// TIA Portal project "Oefening 9" (V14)

(* hardware
DEVICE "S7300/ET200M station_1"  S7-300 station
   slot 0: "Rail_0"  Rail  6ES7 390-1***0-0AA0
   slot 1: "PS 307 10A_1"  PS 307 10A  6ES7 307-1KA02-0AA0
   slot 2: "PLC_1"  CPU 314C-2 PN/DP  6ES7 314-6EH04-0AB0  V3.3
      slot 2: "PROFINET interface_1"  PN-IO
         slot 1: "Port_1"  Port
         slot 2: "Port_2"  Port
      slot 5: "DI 24/DO 16_1"  DI24/DO16
      slot 6: "AI 5/AO 2_1"  AI5/AO2
      slot 7: "Count_1"  Counter
      slot 8: "Positioning_1"  Positioning
   slot 4: "DI 16/DO 16x24VDC/0.5A_1"  DI16/DO16 x 24V / 0.5A  6ES7 323-1BL00-0AA0
*)

// ===== PLC "PLC_1"  CPU 314C-2 PN/DP =====

VAR_GLOBAL   // PLC tag table "Default tag table"
   "S10" AT %I136.0 : Bool;
   "S11" AT %I136.1 : Bool;
   "S12" AT %I136.2 : Bool;
   "S13" AT %I136.3 : Bool;
   "S14" AT %I136.4 : Bool;
   "S15" AT %I136.5 : Bool;
   "S16" AT %I136.6 : Bool;
   "S17" AT %I136.7 : Bool;
   "S0" AT %I138.0 : Bool;
   "S1" AT %I138.1 : Bool;
   "S2" AT %I138.2 : Bool;
   "S3" AT %I138.3 : Bool;
   "S4" AT %I138.4 : Bool;
   "S5" AT %I138.5 : Bool;
   "S6" AT %I138.6 : Bool;
   "S7" AT %I138.7 : Bool;
   "Lre1" AT %Q136.0 : Bool;
   "Lor1" AT %Q136.1 : Bool;
   "Lgr1" AT %Q136.2 : Bool;
   "Lre2" AT %Q136.3 : Bool;
   "Lor2" AT %Q136.4 : Bool;
   "Lgr2" AT %Q136.5 : Bool;
   "Lbl" AT %Q136.6 : Bool;
   "Lwh" AT %Q136.7 : Bool;
   "Pot" AT %IW800 : Int;
   "Emergency" AT %I1.7 : Bool;
   "diD1" AT %MD54 : DInt;
   "diD2" AT %MD58 : DInt;
   "diE1" AT %MD74 : DInt;
   "diE2" AT %MD78 : DInt;
   "iD1" AT %MW50 : Int;
   "iD2" AT %MW52 : Int;
   "iE1" AT %MW70 : Int;
   "iE2" AT %MW72 : Int;
   "iI1" AT %MW90 : Int;
   "iI2" AT %MW92 : Int;
   "iI3" AT %MW94 : Int;
   "iS1" AT %MW96 : Int;
   "iS2" AT %MW98 : Int;
   "k1" AT %M102.0 : Bool;
   "k2" AT %M102.1 : Bool;
   "k11" AT %M103.2 : Bool;
   "k12" AT %M103.3 : Bool;
   "k13" AT %M103.4 : Bool;
   "k14" AT %M103.5 : Bool;
   "k15" AT %M103.6 : Bool;
   "k16" AT %M103.7 : Bool;
   "k17" AT %M104.0 : Bool;
   "k18" AT %M104.1 : Bool;
   "k3" AT %M102.2 : Bool;
   "k4" AT %M102.3 : Bool;
   "k5" AT %M102.4 : Bool;
   "k6" AT %M102.5 : Bool;
   "k7" AT %M102.6 : Bool;
   "k8" AT %M102.7 : Bool;
   "k9" AT %M103.0 : Bool;
   "k10" AT %M103.1 : Bool;
   "rD1" AT %MD62 : Real;
   "rD2" AT %MD66 : Real;
   "rE1" AT %MD82 : Real;
   "rE2" AT %MD86 : Real;
   "strM1" AT %MB150 : Char;
   "strM2" AT %MB200 : Char;
   "wD1" AT %MW10 : Word;
   "wD2" AT %MW100 : Word;
   "Tag_1" AT %I126.1 : Bool;
   "Tag_2" AT %M10.0 : Bool;
   "Tag_3" AT %M10.1 : Bool;
END_VAR

FUNCTION "FC_1" : Void   // FC1, FBD
{ S7_Optimized_Access := 'FALSE' }
VERSION : 0.1
BEGIN

REGION Network 1: Start/Stop
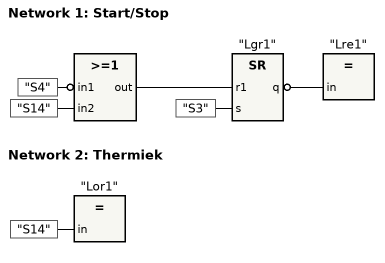
   IF "S3" THEN
       "Lgr1" := TRUE;   // SR flip-flop
   END_IF;
   IF NOT "S4" OR "S14" THEN "Lgr1" := FALSE; END_IF;
   "Lre1" := NOT "Lgr1";
END_REGION

REGION Network 2: Thermiek
   "Lor1" := "S14";
END_REGION
END_FUNCTION

ORGANIZATION_BLOCK "Main"   // OB1, LAD
TITLE = "Main Program Sweep (Cycle)"
{ S7_Optimized_Access := 'FALSE' }
VERSION : 0.1
   VAR_TEMP
      OB1_EV_CLASS : Byte;   // Bits 0-3 = 1 (Coming event), Bits 4-7 = 1 (Event class 1)
      OB1_SCAN_1 : Byte;   // 1 (Cold restart scan 1 of OB 1), 3 (Scan 2-n of OB 1)
      OB1_PRIORITY : Byte;   // Priority of OB Execution
      OB1_OB_NUMBR : Byte;   // 1 (Organization block 1, OB1)
      OB1_RESERVED_1 : Byte;   // Reserved for system
      OB1_RESERVED_2 : Byte;   // Reserved for system
      OB1_PREV_CYCLE : Int;   // Cycle time of previous OB1 scan (milliseconds)
      OB1_MIN_CYCLE : Int;   // Minimum cycle time of OB1 (milliseconds)
      OB1_MAX_CYCLE : Int;   // Maximum cycle time of OB1 (milliseconds)
      OB1_DATE_TIME : Date_And_Time;   // Date and time OB1 started
   END_VAR
BEGIN

REGION Network 1
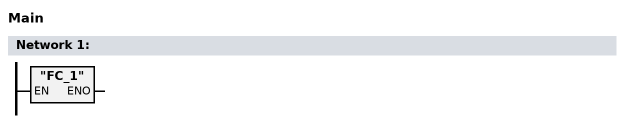
   RUNG wire#powerrail
      "FC_1"()
   END_RUNG
   // the same network as SCL:
   "FC_1"();
END_REGION
END_ORGANIZATION_BLOCK